FUNCTION_BLOCK fbAfstandSensor IMPLEMENTS ITFGesimuleerdAO
VAR_INPUT
END_VAR
VAR_OUTPUT
END_VAR
VAR
	IHmiStackerAfstandSensorSim : INT;
END_VAR

{warning 'Add property implementation'}
PROPERTY SensorWaarde : INT
GET

SensorWaarde := IHmiStackerAfstandSensorSim;
END_GET
SET
IHmiStackerAfstandSensorSim:= SensorWaarde;
END_SET
END_PROPERTY

END_FUNCTION_BLOCK

(* stored: Version 1.1.0.1
   POU fbAfstandSensor: Id {15cf4fdc-c9f7-48c2-9531-7e024c33e696}, SpecialFunc None
   Property SensorWaarde: Id {31f9ff59-3116-4f7c-b92a-04c0c9e91b35}
   Get Get: Id {cff1a2a2-3eb3-4b1f-8005-631fa573ccfe}
   Set Set: Id {e3a6cffd-5cb8-4d70-9c43-fc42aff29e98} *)
